FUNCTION_BLOCK FB_ZoneAggregator IMPLEMENTS I_SafetyZone
VAR
    _eZoneId        : E_ZoneId;
    _stZoneData     : ST_ZoneData;
    _aSlots         : ARRAY[1..30] OF ST_SensorSlot;
    _nSlotCount     : INT := 0;
END_VAR
VAR_INPUT
    eZoneId         : E_ZoneId;
END_VAR

// runs every cycle
// keeps internal zone id in sync with input
_stZoneData.eZoneId := eZoneId;

METHOD CheckSafety : E_ZoneState

THIS^.UpdateSensors();
CheckSafety := _stZoneData.eZoneState;
END_METHOD

METHOD CheckZoneData : ST_ZoneData

CheckZoneData := _stZoneData;
END_METHOD

METHOD GetZoneState : E_ZoneState

GetZoneState := _stZoneData.eZoneState;
END_METHOD

PROPERTY HasAlarm : BOOL
GET
HasAlarm := _stZoneData.eWorstAlarmLevel > E_AlarmLevel.INFO;
END_GET
SET
END_SET
END_PROPERTY

METHOD RegisterH2SSensor :BOOL
VAR_IN_OUT
    fbSensor      : FB_BaseSensor;    // VAR_IN_OUT = reference
END_VAR
VAR
    ipTemp  : I_SafetySensor;
END_VAR

IF _nSlotCount >= 30 THEN
    RegisterH2SSensor := FALSE;
    RETURN;
END_IF

_nSlotCount := _nSlotCount + 1;

ipTemp := fbsensor;
_aSlots[_nSlotCount].ipSensor         := ipTemp;
_aSlots[_nSlotCount].eSensorType      := E_SensorType.H2S;
_aSlots[_nSlotCount].bOccupied        := TRUE;
_aSlots[_nSlotCount].bIsH2SCritical   := TRUE;
_aSlots[_nSlotCount].bIsSmokeCritical := FALSE;

RegisterH2SSensor := TRUE;
END_METHOD

METHOD RegisterSensor : BOOL
VAR_IN_OUT
    fbsensor      : FB_BaseSensor;    // VAR_IN_OUT = reference
END_VAR
VAR_INPUT
    eType       : E_SensorType;
END_VAR
VAR
    ipTemp  : I_SafetySensor;
END_VAR

IF _nSlotCount >= 30 THEN
    RegisterSensor := FALSE;
    RETURN;
END_IF

_nSlotCount := _nSlotCount + 1;

// ✅ CORRECT way in TwinCAT
// assign VAR_IN_OUT reference to interface
// TwinCAT resolves vtable correctly this way
// DO NOT use ADR() for interface assignment
ipTemp := fbsensor;
_aSlots[_nSlotCount].ipSensor         := ipTemp;
_aSlots[_nSlotCount].eSensorType      := eType;
_aSlots[_nSlotCount].bOccupied        := TRUE;
_aSlots[_nSlotCount].bIsH2SCritical   := FALSE;
_aSlots[_nSlotCount].bIsSmokeCritical := FALSE;

RegisterSensor := TRUE;
END_METHOD

METHOD RegisterSmokeSensor : BOOL
VAR_IN_OUT
    fbsensor      : FB_BaseSensor;    // VAR_IN_OUT = reference
END_VAR
VAR
    ipTemp  : I_SafetySensor;
END_VAR
IF _nSlotCount >= 30 THEN
    RegisterSmokeSensor := FALSE;
    RETURN;
END_IF

_nSlotCount := _nSlotCount + 1;

ipTemp := fbsensor;
_aSlots[_nSlotCount].ipSensor         := ipTemp;
_aSlots[_nSlotCount].eSensorType      := E_SensorType.SMOKE;
_aSlots[_nSlotCount].bOccupied        := TRUE;
_aSlots[_nSlotCount].bIsH2SCritical   := FALSE;
_aSlots[_nSlotCount].bIsSmokeCritical := TRUE;

RegisterSmokeSensor := TRUE;
END_METHOD

METHOD Reset : BOOL
VAR
    i : INT;
END_VAR

FOR i := 1 TO _nSlotCount DO
    IF _aSlots[i].bOccupied THEN
        _aSlots[i].ipSensor.Reset();
    END_IF
END_FOR

_stZoneData.eZoneState       := E_ZoneState.ZONE_NORMAL;
_stZoneData.eWorstAlarmLevel := E_AlarmLevel.NONE;
_stZoneData.bESDRequired     := FALSE;
_stZoneData.bH2SAlarm        := FALSE;
Reset := TRUE;
END_METHOD

METHOD TriggerESD : BOOL
VAR_INPUT
    eLevel : E_ESDLevel;
END_VAR
_stZoneData.bESDRequired := TRUE;
_stZoneData.eZoneState   := E_ZoneState.ZONE_EMERGENCY;
TriggerESD := TRUE;
END_METHOD

METHOD UpdateSensors 
VAR
    i            : INT;
    nAlarms      : INT;
    nGasAlarms   : INT;
    nPressAlarms : INT;
    nTempAlarms  : INT;
    bH2SAlarm    : BOOL;
    bSmokeAlarm  : BOOL;
    bAnyAlarm    : BOOL;
END_VAR

i            := 0;
nAlarms      := 0;
nGasAlarms   := 0;
nPressAlarms := 0;
nTempAlarms  := 0;
bH2SAlarm    := FALSE;
bSmokeAlarm  := FALSE;
bAnyAlarm    := FALSE;

// ─────────────────────────────────────
// Pass 1 — H2S
// ─────────────────────────────────────
FOR i := 1 TO _nSlotCount DO
    IF _aSlots[i].bOccupied
       AND _aSlots[i].bIsH2SCritical
       AND _aSlots[i].ipSensor <> 0 THEN    // ✅ null check
        IF _aSlots[i].ipSensor.IsAlarm() THEN
            bH2SAlarm := TRUE;
        END_IF
    END_IF
END_FOR

// ─────────────────────────────────────
// Pass 2 — Smoke
// ─────────────────────────────────────
FOR i := 1 TO _nSlotCount DO
    IF _aSlots[i].bOccupied
       AND _aSlots[i].bIsSmokeCritical
       AND _aSlots[i].ipSensor <> 0 THEN    // ✅ null check
        IF _aSlots[i].ipSensor.IsAlarm() THEN
            bSmokeAlarm := TRUE;
        END_IF
    END_IF
END_FOR

// ─────────────────────────────────────
// Pass 3 — standard sensors vote count
// ─────────────────────────────────────
FOR i := 1 TO _nSlotCount DO
    IF _aSlots[i].bOccupied
       AND NOT _aSlots[i].bIsH2SCritical
       AND NOT _aSlots[i].bIsSmokeCritical
       AND _aSlots[i].ipSensor <> 0 THEN    // ✅ null check
        IF _aSlots[i].ipSensor.IsAlarm() THEN
            nAlarms   := nAlarms + 1;
            bAnyAlarm := TRUE;
            CASE _aSlots[i].eSensorType OF
                E_SensorType.GAS:
                    nGasAlarms := nGasAlarms + 1;
                E_SensorType.PRESSURE:
                    nPressAlarms := nPressAlarms + 1;
                E_SensorType.TEMP:
                    nTempAlarms := nTempAlarms + 1;
            END_CASE
        END_IF
    END_IF
END_FOR

// ─────────────────────────────────────
// Write all counts before voting
// ─────────────────────────────────────
_stZoneData.eZoneId             := eZoneId;
_stZoneData.bH2SAlarm           := bH2SAlarm;
_stZoneData.nGasAlarmCount      := nGasAlarms;
_stZoneData.nPressureAlarmCount := nPressAlarms;
_stZoneData.nTempAlarmCount     := nTempAlarms;
_stZoneData.tLastUpdate         := TIME();

IF bAnyAlarm OR bH2SAlarm OR bSmokeAlarm THEN
    _stZoneData.tLastAlarm := TIME();
END_IF

// ─────────────────────────────────────
// Voting logic
// ─────────────────────────────────────
IF bH2SAlarm OR bSmokeAlarm THEN
    _stZoneData.eWorstAlarmLevel := E_AlarmLevel.CRITICAL;
    _stZoneData.eZoneState       := E_ZoneState.ZONE_EMERGENCY;
    _stZoneData.bESDRequired     := TRUE;
    _stZoneData.sStatusMessage   := 'EMERGENCY - H2S or Smoke';

ELSIF nAlarms >= GVL_SafetyLimits.c_nVOTE_EMERGENCY THEN
    _stZoneData.eWorstAlarmLevel := E_AlarmLevel.CRITICAL;
    _stZoneData.eZoneState       := E_ZoneState.ZONE_EMERGENCY;
    _stZoneData.bESDRequired     := TRUE;
    _stZoneData.sStatusMessage   := 'EMERGENCY - ESD required';

ELSIF nAlarms >= GVL_SafetyLimits.c_nVOTE_WARNING THEN
    _stZoneData.eWorstAlarmLevel := E_AlarmLevel.WARNING;
    _stZoneData.eZoneState       := E_ZoneState.ZONE_WARNING;
    _stZoneData.bESDRequired     := FALSE;
    _stZoneData.sStatusMessage   := 'WARNING - operator action required';

ELSIF nAlarms >= GVL_SafetyLimits.c_nVOTE_ALERT THEN
    _stZoneData.eWorstAlarmLevel := E_AlarmLevel.INFO;
    _stZoneData.eZoneState       := E_ZoneState.ZONE_ALERT;
    _stZoneData.bESDRequired     := FALSE;
    _stZoneData.sStatusMessage   := 'ALERT - investigate sensor';

ELSE
    _stZoneData.eWorstAlarmLevel := E_AlarmLevel.NONE;
    _stZoneData.eZoneState       := E_ZoneState.ZONE_NORMAL;
    _stZoneData.bESDRequired     := FALSE;
    _stZoneData.sStatusMessage   := 'NORMAL - all sensors ok';
END_IF
END_METHOD

PROPERTY  ZoneData : ST_ZoneData
GET
ZoneData := _stZoneData;
END_GET
SET
END_SET
END_PROPERTY

PROPERTY ZoneState : E_ZoneState
GET
ZoneState := _stZoneData.eZoneState;
END_GET
SET
END_SET
END_PROPERTY

END_FUNCTION_BLOCK

(* stored: Version 1.1.0.1, ProductVersion 3.1.4024.16
   POU FB_ZoneAggregator: Id {6cdb20ee-13d7-4f10-9fef-8b030c5d2fac}, SpecialFunc None
   Method CheckSafety: Id {00db5e66-ee6d-41ae-9e7a-987f5949bf52}
   Method CheckZoneData: Id {f3f3d24d-1a2b-4789-a4bc-b8b834377581}
   Method GetZoneState: Id {2288b829-db5c-491f-876f-212c6cda2a9c}
   Property HasAlarm: Id {651f0b9d-e765-46b1-827c-320315888fc8}
   Get Get: Id {bdbe05e6-66fb-4441-8d00-583f6506e453}
   Set Set: Id {a9ee90e1-882b-4040-b098-a3f5e2b4b4d4}
   Method RegisterH2SSensor: Id {f22b822c-d766-46a9-a14a-8cba8fe79201}
   Method RegisterSensor: Id {8ebde41c-833c-49d1-8e46-aa849dd3e43c}
   Method RegisterSmokeSensor: Id {5cf2fa83-cbb0-4084-9e21-2755b472f7be}
   Method Reset: Id {8e5cfc46-807d-47f9-834e-29a633e04435}
   Method TriggerESD: Id {955c0f99-7a47-4fc7-92e4-b43787744cba}
   Method UpdateSensors: Id {c3d76990-c668-46d5-9002-6f41123b0859}
   Property ZoneData: Id {a4a93b7c-e9fa-43d2-9970-d3459a260641}
   Get Get: Id {a5e4dd85-5a52-421c-8f5a-fbb30f5bc670}
   Set Set: Id {0c3c2426-7877-417b-a671-2d0d755105e8}
   Property ZoneState: Id {e5ad2492-60ac-4890-8235-e0bec85b225e}
   Get Get: Id {336e8d7c-0d8d-4914-9340-b2f24197fa2f}
   Set Set: Id {9ba6dd5b-7dda-47fd-8f80-3f7d71346363} *)
